Staubli VAL3: show_data.pgx

public program show_data()
begin

   do
    cls()
    put("Reference Velocity [mm/s]: ")
    put(Ref_Vel)
    putln("")
    //cls()
    put("Robot Velocity [mm/s]: ")
    put(getSpeed(tTool))
    putln("")
    //cls()
    put("Error (Ref-Rob) [mm/s]: ")
    put(Ref_Vel - getSpeed(tTool))
    putln("")
    //cls()
    put("Current position: ")
    put(getMoveId())
    putln("")


    delay(0.001)
    //putln("")
  until check_status != true

end
